(* Logix 5000 project; controller PLC2_Project_8 Emulate 5570 rev 20.11; software revision 20.00 *)
// PID substitution logic

TASK MainTask (continuous, watchdog 500 ms) : MainProgram

MODULES
   Local : Emulate 5570 (ICP 1, rev 20.11)
END_MODULES

ADD_ON_INSTRUCTION NSCP   (* revision 1.0 *)
// Nicks Scale With Parameters
VAR_INPUT
   InputMax : DINT; {required}
   InputMin : DINT; {required}
   ScaledMaxOut : DINT; {required}
   ScaledMinOut : DINT; {required}
   Input : DINT; {required}
END_VAR
VAR_OUTPUT
   ScaledOutput : REAL; {access Read Only, required}
END_VAR
VAR
   Rate : REAL; {access None}
END_VAR

ROUTINE Logic   (* structured text *)
   // My scale with parameters
   IF (EnableIn) THEN
   	Rate := (ScaledMaxOut - ScaledMinOut) / (InputMax - InputMin);
   	ScaledOutput := (Input - InputMin) * Rate + ScaledMinOut;
   END_IF;
END_ROUTINE
END_ADD_ON_INSTRUCTION

PROGRAM MainProgram   (* main routine _00_Main *)
VAR
   _sim_eq : REAL; {access Read Only}
   _sim_sensor_output_scaled : REAL; {access Read Only}
   _sim_sensor_output_SCP : NSCP; {access Read Only}
   _sim_sensor_raw_systemInput : DINT; {access Read Only}
   _sim_Timer : FBD_TIMER; {access Read Only}
   _sim_vfd_en : BOOL; {access Read Only}
   _sim_vfd_input_scaled : REAL; {access Read Only}
   _sim_vfd_input_SCP : NSCP; {access Read Only}
   _sim_vfd_raw_systemOutput : DINT; {access Read Only}
   _sim_x : REAL; {access Read Only}
   InHg_DiffAbs : REAL; {access Read Only}
   InHg_Difference : REAL; {access Read Only}
   InHg_Range_1 : REAL; {access Read Only}   // 1
   InHg_Range_2 : REAL; {access Read Only}   // 2
   InHg_Range_3 : REAL; {access Read Only}   // 5
   InHg_Range_4 : REAL; {access Read Only}   // 7
   InHg_SetPoint : REAL; {access Read Only}
   Sensor_INHG_In_Scaled : REAL; {access Read Only}
   Sensor_Input_NSCP : NSCP; {access Read Only}
   Vfd_En : BOOL; {access Read Only}
   Vfd_Out_Pct : REAL; {access Read Only}
   Vfd_Output_NSCP : NSCP; {access Read Only}
   Vfd_Start : BOOL; {access Read Only}
   Vfd_Stop : BOOL; {access Read Only}
END_VAR

ROUTINE _00_Main   (* ladder *)
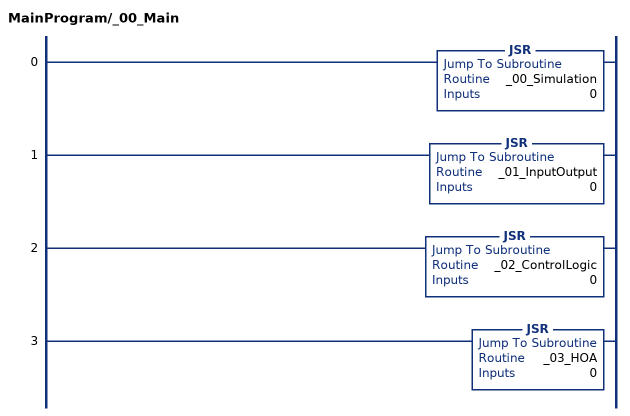
   0: JSR(_00_Simulation,0);
   1: JSR(_01_InputOutput,0);
   2: JSR(_02_ControlLogic,0);
   3: JSR(_03_HOA,0);
END_ROUTINE

ROUTINE _00_Simulation   (* structured text *)
// Vacuum chamber simulation. Changes with time.
   _sim_Timer.PRE := 100;
   _sim_Timer.TimerEnable :=1;
   TONR(_sim_Timer);
   
   // Put sim logic here
   IF (_sim_Timer.DN) THEN
   	_sim_x := _sim_x + 0.1;
   END_IF;
   
   // If the vfd/pump (combine them for simplicity) is turned on:
   IF (_sim_vfd_en) THEN
   	_sim_vfd_raw_systemOutput := 8419;
   
   	// Scale the input sensor values into something we can work with:
   	_sim_vfd_input_SCP.EnableIn := 1;
   	NSCP(_sim_vfd_input_SCP, 16383, 0, 50, -50, _sim_vfd_raw_systemOutput, _sim_vfd_input_scaled);
   
   	// Equation to simulate changing environment.
   	//
   	_sim_sensor_output_scaled := 6.0 * sin(0.8*_sim_x) + 3.0 * sin(2.0 * _sim_x) + 15.0 - _sim_vfd_input_scaled / 3.0;
   
   	IF (_sim_sensor_output_scaled >= 30) THEN
   		_sim_sensor_output_scaled := 30;
   	END_IF;
   
   	IF (_sim_sensor_output_scaled <= 0) THEN
   		_sim_sensor_output_scaled := 0;
   	END_IF;
   END_IF;
   
   // If the vfd/pump (combine them for simplicity) is turned off
   IF NOT (_sim_vfd_en) THEN
   	_sim_sensor_output_scaled := 30;
   END_IF;
   
   // Scale the output sensor values:
   _sim_sensor_raw_systemInput := _sim_sensor_output_SCP.ScaledOutput;
   NSCP(_sim_sensor_output_SCP, 0, 30, 16383, 0, _sim_sensor_output_scaled, _sim_sensor_raw_systemInput);
   
   // End sim logic
   _sim_Timer.Reset := _sim_Timer.DN;
END_ROUTINE

ROUTINE _01_InputOutput   (* ladder *)
// Inputs & Outputs
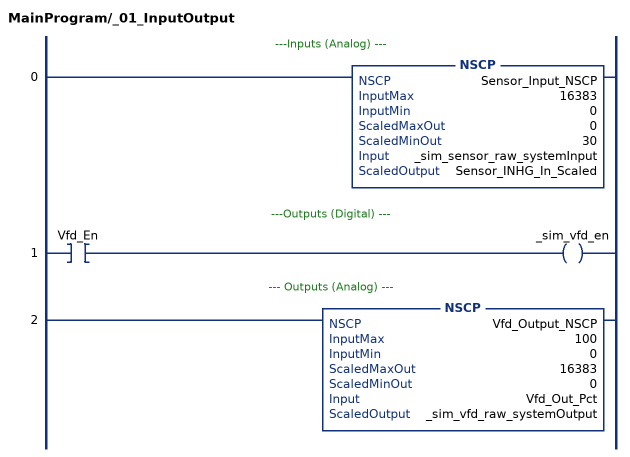
   // ---Inputs (Analog) ---
   0: NSCP(Sensor_Input_NSCP,16383,0,0,30,_sim_sensor_raw_systemInput,Sensor_INHG_In_Scaled);
   // ---Outputs (Digital) ---
   1: XIC(Vfd_En)OTE(_sim_vfd_en);
   // --- Outputs (Analog) ---
   2: NSCP(Vfd_Output_NSCP,100,0,16383,0,Vfd_Out_Pct,_sim_vfd_raw_systemOutput);
END_ROUTINE

ROUTINE _02_ControlLogic   (* ladder *)
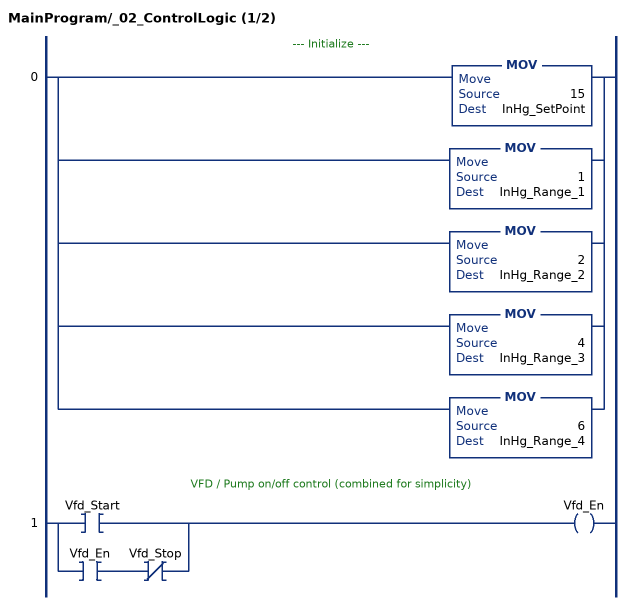
   // --- Initialize ---
   0: [MOV(15,InHg_SetPoint) ,MOV(1,InHg_Range_1) ,MOV(2,InHg_Range_2) ,MOV(4,InHg_Range_3) ,MOV(6,InHg_Range_4) ];
   // VFD / Pump on/off control (combined for simplicity)
   1: [XIC(Vfd_Start) ,XIC(Vfd_En) XIO(Vfd_Stop) ]OTE(Vfd_En);
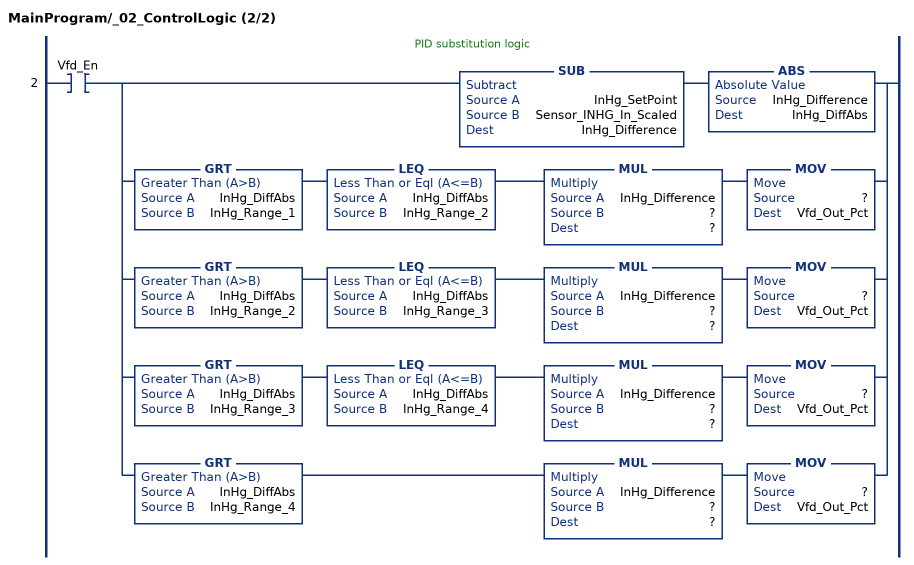
   // PID substitution logic
   2: XIC(Vfd_En)[SUB(InHg_SetPoint,Sensor_INHG_In_Scaled,InHg_Difference) ABS(InHg_Difference,InHg_DiffAbs) ,GRT(InHg_DiffAbs,InHg_Range_1) LEQ(InHg_DiffAbs,InHg_Range_2) MUL(InHg_Difference,?,?) MOV(?,Vfd_Out_Pct) ,GRT(InHg_DiffAbs,InHg_Range_2) LEQ(InHg_DiffAbs,InHg_Range_3) MUL(InHg_Difference,?,?) MOV(?,Vfd_Out_Pct) ,GRT(InHg_DiffAbs,InHg_Range_3) LEQ(InHg_DiffAbs,InHg_Range_4) MUL(InHg_Difference,?,?) MOV(?,Vfd_Out_Pct) ,GRT(InHg_DiffAbs,InHg_Range_4) MUL(InHg_Difference,?,?) MOV(?,Vfd_Out_Pct) ];
END_ROUTINE

ROUTINE _03_HOA   (* ladder *)
// Hand-Off-Auto
   0: ;
END_ROUTINE
END_PROGRAM
